{attribute addProperty BoxType "EL6688-0000-0017"}
{attribute addProperty Id "External_SyncAT %I*External_Sync_AA57C188192240WcStateAT %I*WcState_F855686C1620InfoDataAT %I*InfoData_0BDED7BF144180"}
{attribute addProperty CRC "1599302842"}
{attribute addProperty SizeInBites "352"}
{attribute addProperty SizeInBytes "44"}
TYPE EL6688_8282893D :
STRUCT
	{attribute addProperty Name "External_Sync"}
	External_Sync : External_Sync_AA57C188;
	{attribute addProperty Name "WcState"}
	WcState : WcState_F855686C;
	{attribute addProperty Name "InfoData"}
	InfoData : InfoData_0BDED7BF;
END_STRUCT
END_TYPE

(* stored: Version 1.2.0.0, ProductVersion 3.1.4024.9
   DUT EL6688_8282893D: Id {5a58835f-53d4-49ad-abb0-7357fa45954b} *)
